FUNCTION_BLOCK PLOT2D_SCATTER
  {SET_ATTRIBUTE(OpcUa, SERVICE)}
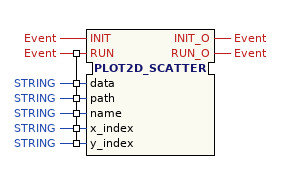
  EVENT_INPUT
    INIT;
    RUN WITH data, path, name, x_index, y_index; {SET_ATTRIBUTE(OpcUa, Method)}
  END_EVENT
  EVENT_OUTPUT
    INIT_O;
    RUN_O;
  END_EVENT
  VAR_INPUT
    data : STRING; {SET_ATTRIBUTE(OpcUa, Variable)}
    path : STRING; {SET_ATTRIBUTE(OpcUa, Variable)}
    name : STRING; {SET_ATTRIBUTE(OpcUa, Variable)}
    x_index : STRING; {SET_ATTRIBUTE(OpcUa, Variable)}
    y_index : STRING; {SET_ATTRIBUTE(OpcUa, Variable)}
  END_VAR
END_FUNCTION_BLOCK
